(* PLC project  *)

CONFIGURATION FSLOGIC_1
END_CONFIGURATION
